SUBAPPLICATION mapping_Uebung_025 (* Spiegelabfolge (5) *)
  (* Standard: 61499-2; Description: Copyright (c) 2023 Meisterschulen am Ostbahnhof This program and the accompanying materials are made available under the terms of the Eclipse Public License 2.0 which is available at https://www.eclipse.org/legal/epl-2.0/ SPDX-License-Identifier: EPL-2.0 *)
  (* Version 1.0, 2023-10-23, Franz Höpfinger, Meisterschulen am Ostbahnhof *)
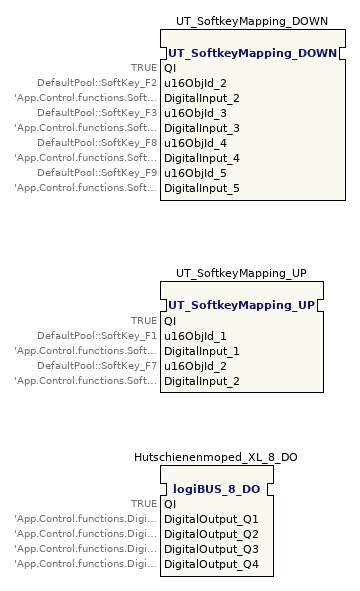
  FBS
    Hutschienenmoped_XL_8_DO : logiBUS_8_DO(QI := TRUE, DigitalOutput_Q1 := 'App.Control.functions.DigitalOutput_Q1', DigitalOutput_Q2 := 'App.Control.functions.DigitalOutput_Q2', DigitalOutput_Q3 := 'App.Control.functions.DigitalOutput_Q3', DigitalOutput_Q4 := 'App.Control.functions.DigitalOutput_Q4');
    UT_SoftkeyMapping_UP : UT_SoftkeyMapping_UP(QI := TRUE, u16ObjId_1 := DefaultPool::SoftKey_F1, DigitalInput_1 := 'App.Control.functions.SoftKey_F1_UP', u16ObjId_2 := DefaultPool::SoftKey_F7, DigitalInput_2 := 'App.Control.functions.SoftKey_F7_UP');
    UT_SoftkeyMapping_DOWN : UT_SoftkeyMapping_DOWN(QI := TRUE, u16ObjId_2 := DefaultPool::SoftKey_F2, DigitalInput_2 := 'App.Control.functions.SoftKey_F2_DOWN', u16ObjId_3 := DefaultPool::SoftKey_F3, DigitalInput_3 := 'App.Control.functions.SoftKey_F3_DOWN', u16ObjId_4 := DefaultPool::SoftKey_F8, DigitalInput_4 := 'App.Control.functions.SoftKey_F8_DOWN', u16ObjId_5 := DefaultPool::SoftKey_F9, DigitalInput_5 := 'App.Control.functions.SoftKey_F9_DOWN');
  END_FBS
END_SUBAPPLICATION
